{attribute addProperty BoxType "EPP2624-0002-0016"}
{attribute addProperty Id "ChannelAT %Q*ARRAY[0..3] OF Channel_7F374EB03240WcStateAT %I*WcState_28A8677510.1250InfoDataAT %I*InfoData_192954DE1620"}
{attribute addProperty CRC "2753798610"}
{attribute addProperty SizeInBites "49"}
{attribute addProperty SizeInBytes "6.125"}
TYPE EPP2624_4E3C7537 :
STRUCT
	{attribute addProperty Name "Channel"}
	Channel : ARRAY[0..3] OF Channel_7F374EB0;
	{attribute addProperty Name "WcState"}
	WcState : WcState_28A86775;
	{attribute addProperty Name "InfoData"}
	InfoData : InfoData_192954DE;
END_STRUCT
END_TYPE

(* stored: Version 1.2.0.0, ProductVersion 3.1.4024.9
   DUT EPP2624_4E3C7537: Id {cb3611a3-7c20-4e88-b011-afb454ef7198} *)
